INTERFACE ITF_Component_TE1_HMI_Init EXTENDS ITF_BaseComponent, ITF_Component_TE1_HMI_Connector

END_INTERFACE

(* stored: Version 1.1.0.1, ProductVersion 3.1.4024.15
   Itf ITF_Component_TE1_HMI_Init: Id {ba80b561-9bc9-4971-aa2c-d7234bf19f42} *)
